{attribute 'qualified_only'}
{attribute 'strict'}
TYPE PathfindingResult :
(
	valid := 0,
	error,
	notNeeded
);
END_TYPE

(* stored: Version 1.1.0.1, ProductVersion 3.1.4024.11
   DUT PathfindingResult: Id {13366d8a-29e6-4cf8-9518-0305767f0d7d} *)
